// TIA Portal V20 export
DATA_BLOCK "ComRd"   // DB361
{ S7_Optimized_Access := 'FALSE' }
// stored: AutoNumber false
   VAR
      Plc : "TypeHeaderPlc";   // Header Plc
      Pc : "TypeHeaderPcGld";   // Header Pc
      Data : Struct
         Config : Struct   // config
            "version" : Int;   // version info
            active : Bool;   // config active (Test Output not active)
            adjScannerActive : Bool;   // adjustment scanner housing active
            adjTopActive : Bool;   // adjustment metering bar top active
            adjLeftActive : Bool;   // adjustment metering bar left active
            adjRightActive : Bool;   // adjustment metering bar right active
            adjTopLinMotActive : Bool;   // adjustment metering bar top active - linear drive
            adjLeftLinMotActive : Bool;   // adjustment metering bar left active - linear drive
            adjRightLinMotActive : Bool;   // adjustment metering bar right active - linear drive
            xrayActive : Bool;   // xray active
            adjLaserTopLeftStepMotActive : Bool;   // adjustment laser top left active - step motor
            adjLaserTopRightStepMotActive : Bool;   // adjustment laser top right active - step motor
            adjLaserLeftTopStepMotActive : Bool;   // adjustment laser left top active - step motor
            adjLaserLeftBottomStepMotActive : Bool;   // adjustment laser left bottom active - step motor
            adjLaserRightTopStepMotActive : Bool;   // adjustment laser right top active - step motor
            adjLaserRightBottomStepMotActive : Bool;   // adjustment laser right bottom active - step motor
            modeBoardPassing : Int;   // 1=left / 2=rigth / 3=middle
            modeDimension : Int;   // 1=fixed / 2=random width / 3=random thickness / 4=random width + thickness
            modeRandomAdj : Int;   // 1=with sensor / 2=with external data
            spare40 : Int;   // spare
            spare42 : Int;   // spare
            enc1Factor : Int;   // encoder infeed factor
            spare46 : Int;   // spare
            spare48 : Int;   // spare
            enc1QuadEvalActive : Bool;   // encoder infeed - quadruple evaluation active
            spare501 : Bool;   // spare
            spare502 : Bool;   // spare
         END_STRUCT;
         control : Struct   // control
            spare1 : Bool;
            spare2 : Bool;
         END_STRUCT;
         safety : Struct   // safety
            AreaLaserOn : Bool;   // area laser on
            AreaAdjustmentOn : Bool;   // area adjustment on
            AreaXrayOn : Bool;   // area X-Ray on
            ResetSafetyDevice : Bool;   // reset safety device
         END_STRUCT;
         status : Struct   // status
            Auto : Bool;   // automatic mode scanner
            StopFeeding : Bool;   // stop feeding scanner (error active)
         END_STRUCT;
         batch : Struct   // batch info
            MinWidth : DInt;   // min width [mm/10]
            MaxWidth : DInt;   // max width [mm/10]
            MinThickness : DInt;   // min thickness [mm/10]
            MaxThickness : DInt;   // max thickness [mm/10]
         END_STRUCT;
         Scanner : "TypeAxisRd";   // adjustment scanner
         Top : "TypeAxisRd";   // adjustment top
         Left : "TypeAxisRd";   // adjustment left
         Right : "TypeAxisRd";   // adjustment right
         Measure : Struct   // measuring sensor for random width/thickness
            SetCalibratePosTop : Bool;   // set calibrated position for sensor top
            SetCalibratePosLeft : Bool;   // set calibrated position for sensor left
            SetCalibratePosRight : Bool;   // set calibrated position for sensor right
         END_STRUCT;
         TestOutput : Struct   // test output
            Active : Bool;   // test output active
            "Q0.0" : Bool;
            "Q0.1" : Bool;
            "Q0.2" : Bool;
            "Q0.3" : Bool;
            "Q0.4" : Bool;
            "Q0.5" : Bool;
            "Q0.6" : Bool;
            "Q0.7" : Bool;
            "Q1.0" : Bool;
            "Q1.1" : Bool;
            "Q2.0" : Bool;
            "Q2.3" : Bool;
            "Q2.4" : Bool;
            "Q2.5" : Bool;
            "Q2.6" : Bool;
            "Q900.1" : Bool;
            "Q908.0" : Bool;
            "Q908.1" : Bool;
         END_STRUCT;
         res : Array[1..200] of Byte;
      END_STRUCT;
   END_VAR
BEGIN
END_DATA_BLOCK
